% RSLogix 500 project I2P-Job13B-Adam Boczkiewicz.RSS, saved by version 10.00.00.00 %
PROJECT "ML04A"    % processor: Bul.1763 MicroLogix 1100 Series B %

PROGRAM FILES
  LAD 2   12 rungs

DATA FILES
  O0 OUTPUT  4 elements
  I1 INPUT  6 elements
  S2 STATUS  66 elements
  B3 BINARY  1 elements
  T4 TIMER  1 elements
  C5 COUNTER  1 elements
  R6 CONTROL  1 elements
  N7 INTEGER  1 elements
  F8 FLOAT  1 elements

LADDER 2
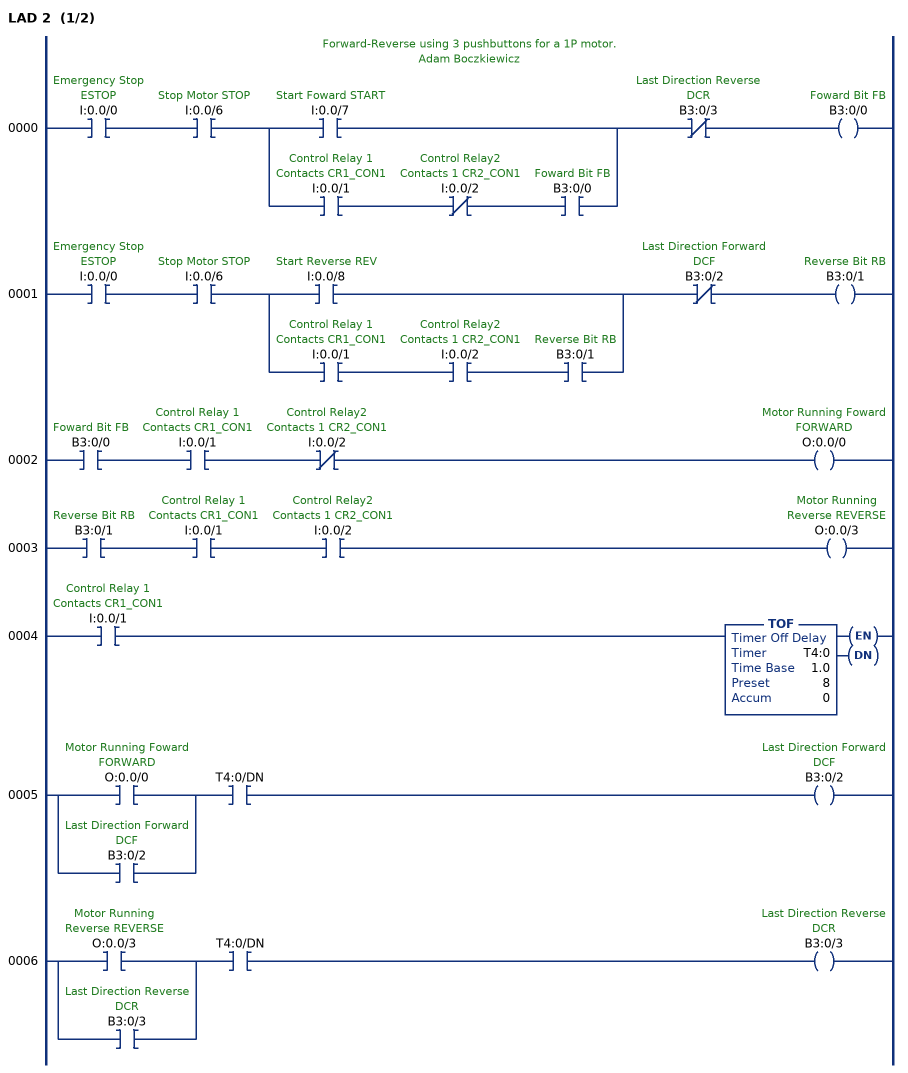
% Rung: 0 %
% Forward-Reverse using 3 pushbuttons for a 1P motor.
% Adam Boczkiewicz %
SOR XIC I:0.0/0 XIC I:0.0/6 BST XIC I:0.0/7 NXB XIC I:0.0/1 XIO I:0.0/2 XIC B3:0/0 BND XIO B3:0/3 OTE B3:0/0 EOR
%   I:0.0/0  ESTOP  "Emergency Stop" %
%   I:0.0/6  STOP  "Stop Motor" %
%   I:0.0/7  START  "Start Foward" %
%   I:0.0/1  CR1_CON1  "Control Relay 1 Contacts" %
%   I:0.0/2  CR2_CON1  "Control Relay2 Contacts 1" %
%   B3:0/0  FB  "Foward Bit" %
%   B3:0/3  DCR  "Last Direction Reverse" %
% Rung: 1 %
SOR XIC I:0.0/0 XIC I:0.0/6 BST XIC I:0.0/8 NXB XIC I:0.0/1 XIC I:0.0/2 XIC B3:0/1 BND XIO B3:0/2 OTE B3:0/1 EOR
%   I:0.0/0  ESTOP  "Emergency Stop" %
%   I:0.0/6  STOP  "Stop Motor" %
%   I:0.0/8  REV  "Start Reverse" %
%   I:0.0/1  CR1_CON1  "Control Relay 1 Contacts" %
%   I:0.0/2  CR2_CON1  "Control Relay2 Contacts 1" %
%   B3:0/1  RB  "Reverse Bit" %
%   B3:0/2  DCF  "Last Direction Forward" %
% Rung: 2 %
SOR XIC B3:0/0 XIC I:0.0/1 XIO I:0.0/2 OTE O:0.0/0 EOR
%   B3:0/0  FB  "Foward Bit" %
%   I:0.0/1  CR1_CON1  "Control Relay 1 Contacts" %
%   I:0.0/2  CR2_CON1  "Control Relay2 Contacts 1" %
%   O:0.0/0  FORWARD  "Motor Running Foward" %
% Rung: 3 %
SOR XIC B3:0/1 XIC I:0.0/1 XIC I:0.0/2 OTE O:0.0/3 EOR
%   B3:0/1  RB  "Reverse Bit" %
%   I:0.0/1  CR1_CON1  "Control Relay 1 Contacts" %
%   I:0.0/2  CR2_CON1  "Control Relay2 Contacts 1" %
%   O:0.0/3  REVERSE  "Motor Running Reverse" %
% Rung: 4 %
SOR XIC I:0.0/1 TOF T4:0 1.0 8 0 EOR
%   I:0.0/1  CR1_CON1  "Control Relay 1 Contacts" %
% Rung: 5 %
SOR BST XIC O:0.0/0 NXB XIC B3:0/2 BND XIC T4:0/DN OTE B3:0/2 EOR
%   O:0.0/0  FORWARD  "Motor Running Foward" %
%   B3:0/2  DCF  "Last Direction Forward" %
% Rung: 6 %
SOR BST XIC O:0.0/3 NXB XIC B3:0/3 BND XIC T4:0/DN OTE B3:0/3 EOR
%   O:0.0/3  REVERSE  "Motor Running Reverse" %
%   B3:0/3  DCR  "Last Direction Reverse" %

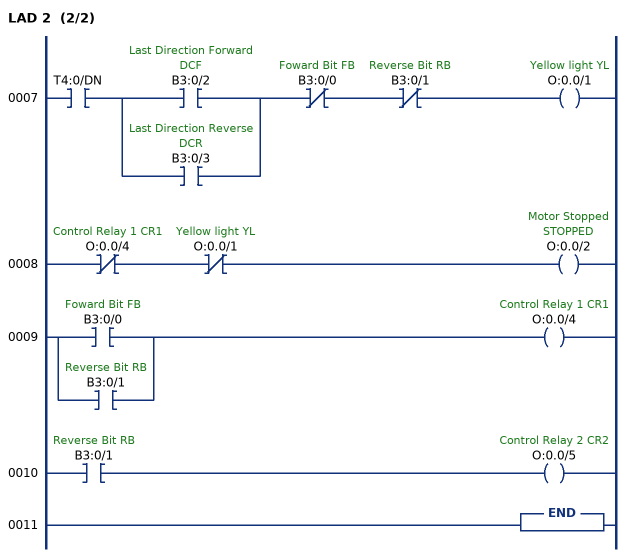
% Rung: 7 %
SOR XIC T4:0/DN BST XIC B3:0/2 NXB XIC B3:0/3 BND XIO B3:0/0 XIO B3:0/1 OTE O:0.0/1 EOR
%   B3:0/2  DCF  "Last Direction Forward" %
%   B3:0/3  DCR  "Last Direction Reverse" %
%   B3:0/0  FB  "Foward Bit" %
%   B3:0/1  RB  "Reverse Bit" %
%   O:0.0/1  YL  "Yellow light" %
% Rung: 8 %
SOR XIO O:0.0/4 XIO O:0.0/1 OTE O:0.0/2 EOR
%   O:0.0/4  CR1  "Control Relay 1" %
%   O:0.0/1  YL  "Yellow light" %
%   O:0.0/2  STOPPED  "Motor Stopped" %
% Rung: 9 %
SOR BST XIC B3:0/0 NXB XIC B3:0/1 BND OTE O:0.0/4 EOR
%   B3:0/0  FB  "Foward Bit" %
%   B3:0/1  RB  "Reverse Bit" %
%   O:0.0/4  CR1  "Control Relay 1" %
% Rung: 10 %
SOR XIC B3:0/1 OTE O:0.0/5 EOR
%   B3:0/1  RB  "Reverse Bit" %
%   O:0.0/5  CR2  "Control Relay 2" %
% Rung: 11 %
SOR END EOR

OTHER DOCUMENTED ADDRESSES
  I:0.0/3  DIRECTION  "Direction:Forward- off-reverse"
  I:0.0/4  DIRECTION_  "Direction: Forward- Off-Reverse"
  I:0.0/5  2PSS  "2 Position Selector Switch"
  T4:0/TT  TT

DATA TABLE (non-zero values as saved)
DATA T4
% .PRE .ACC %
% T4:0 % 8 0
